TYPE FRACTION :
STRUCT
	NUMERATOR : INT;
	DENOMINATOR : INT;
END_STRUCT
END_TYPE

(* stored: Version 1.1.0.1, ProductVersion 3.1.4024.9
   DUT FRACTION: Id {9b46faa7-ec5d-4d12-baaa-dd6df46d99f5} *)
